// TIA Portal V19 export
TYPE "C701_VAR_IF_WMP_TYPIC"
   STRUCT
      REQ_KMO { ExternalAccessible := 'False'; ExternalVisible := 'False'; ExternalWritable := 'False'} : Bool;   // Vrijgave koelmachine bij te hoge koellast
      STO { ExternalAccessible := 'False'; ExternalVisible := 'False'; ExternalWritable := 'False'} : Bool;   // Storing algemeen warmtepomp
   END_STRUCT;
END_TYPE
